{attribute 'GeneratedUsingTerminal: EL6740-0010-0000'}
{attribute addProperty BoxType "EL6740-0010-0000"}
{attribute addProperty Id "StatusAT %I*Status_EF5E6C280InputsEMPTY_STRUCTURE0ControlAT %Q*Control_883019540OutputsEMPTY_STRUCTURE0WcStateAT %I*WcState_9091E0EB2InfoDataAT %I*InfoData_32EB74EA10"}
{attribute addProperty CRC "3140154672"}
{attribute addProperty Size "12"}
TYPE EL6740_BB2AF530 EXTENDS EtcSlaveTerminalBase_947E5A46 :
STRUCT
	{attribute addProperty Name "Status"}
	Status : Status_EF5E6C28;
	{attribute addProperty Name "Inputs"}
	Inputs : EMPTY_STRUCTURE;
	{attribute addProperty Name "Control"}
	Control : Control_88301954;
	{attribute addProperty Name "Outputs"}
	Outputs : EMPTY_STRUCTURE;
	{attribute addProperty Name "WcState"}
	WcState : WcState_9091E0EB;
	{attribute addProperty Name "InfoData"}
	InfoData : InfoData_32EB74EA;
END_STRUCT
END_TYPE

(* stored: Version 1.2.0.0, ProductVersion 3.1.4024.9
   DUT EL6740_BB2AF530: Id {97d7ff48-3703-42f2-894b-49d9178b6bc4} *)
